(* CODESYS project Fiesto_workstation_Biraveen_Nedunchelian.export

Project tree, tasks and I/O mapping:
  Device : CODESYS Control Win V3 x64, 3S - Smart Software Solutions GmbH, version 3.5.16.30
    application Application
      libraries: Standard, * (System)
      task MainTask (cyclic, interval 50 ms, priority 1) calls PLC_PRG
      task VISU_TASK (cyclic, interval 100 ms, priority 31) calls VisuElems.Visu_Prg
      function block Festo_Workstation [ST]
      program PLC_PRG [CFC]
      visualisation Visualization
*)

// Device/Application/PLC_PRG
PROGRAM PLC_PRG
VAR
	Festo: Festo_Workstation;
	lav_indik10: BOOL;
	hoy_indik90: BOOL;
	tanknivaa_tank2: REAL;
	bryter: BOOL;
END_VAR

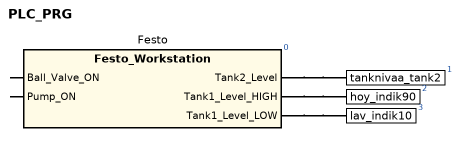
Festo(); // Festo_Workstation
tanknivaa_tank2 := Festo.Tank2_Level;
hoy_indik90 := Festo.Tank1_Level_HIGH;
lav_indik10 := Festo.Tank1_Level_LOW;

END_PROGRAM

// Device/Application/Festo_Workstation
FUNCTION_BLOCK Festo_Workstation
VAR_INPUT
	Ball_Valve_ON : BOOL := FALSE;
	Pump_ON : BOOL := FALSE;
END_VAR
VAR_OUTPUT
	Tank2_Level : REAL := 0;
	Tank1_Level_HIGH : BOOL := TRUE;
	Tank1_Level_LOW : BOOL := TRUE;
END_VAR
VAR
	Inflow : REAL := 0;
	Outflow : REAL := 0;
	Tank1_Level : REAL := 95;
	Inflow_Color : BOOL := FALSE;
	Outflow_Color : BOOL := FALSE;
	Reset : BOOL := FALSE;
	Av_var: REAL;
END_VAR

IF NOT Reset THEN //Reset er FALSE
	IF Pump_ON THEN //Er pumpen på?
		IF Tank1_Level > 0 THEN //Er det noe vann i tank 1? 
			Inflow := 0.2; //Fyll vann i tank 2
			Inflow_Color := TRUE; //Visuvar
		ELSE //Tank 1 er tom
			Inflow := 0; //Ikke fyll
			Inflow_Color := FALSE; //Visuvar
		END_IF
	ELSE //Pumpen er av
		Inflow := 0; //Ikke full
		Inflow_Color := FALSE; //Visuvar
	END_IF
	
	IF Ball_Valve_ON THEN //Er ventilen åpen
		IF Tank2_Level > 0 THEN //Er det vann i tank 2?
			Outflow := 0.1; //Det renner vann tilbake til tank 1
			Outflow_Color := TRUE; //Visuvar
		ELSE //Tank 2 er tom
			Outflow := 0; //Det renner ikke vann
			Outflow_Color := FALSE; //Visuvar
		END_IF
	ELSE //Ventilen er stengt
		Outflow := 0; //Det renner ikke vann
		Outflow_Color := FALSE; //Visuvar
	END_IF
	
	Tank1_Level := Tank1_Level + (Outflow - Inflow); //Level i tank 1
	Tank2_Level := Tank2_Level + (Inflow - Outflow); //Level i tank 2
	
	IF Tank1_Level >= 90 THEN //Er nivået i tank 1 større enn 90?
		Tank1_Level_HIGH := TRUE; //Variabelen er TRUE
	ELSE //Nivået er mindre enn 90
		Tank1_Level_HIGH := FALSE; //Variabel FALSE
	END_IF
	
	IF Tank1_Level <= 10 THEN //Er nivået i tank 1 mindre enn 10?
		Tank1_Level_LOW := FALSE; //Variabel FALSE
	ELSE //Nivået er større enn 10
		Tank1_Level_LOW := TRUE; //Variabel TRUE
	END_IF
ELSE //Reset er TRUE
	//Resetter variablene til initialverdier
	Inflow := 0;
	Outflow := 0;
	Tank1_Level := 95;
	Tank2_Level := 0;
	Tank1_Level_HIGH := FALSE;
	Tank1_Level_LOW := FALSE;
	Pump_ON := FALSE;
	Ball_Valve_ON := FALSE;
	Av_var := 0;
END_IF


IF Tank2_Level > 60 AND Av_var = 0 THEN
	Pump_ON := FALSE;
	Ball_Valve_ON := TRUE;
	Av_var := 1;
END_IF

IF Tank1_Level > 70 AND Av_var = 1 THEN
	Pump_ON := TRUE;
	Ball_Valve_ON := FALSE;
	Av_var := 2;
END_IF

IF Tank2_Level > 10 AND Av_var = 2 THEN
	Ball_Valve_ON := FALSE;
	Pump_ON := TRUE;
	Av_var := 0;
END_IF

END_FUNCTION_BLOCK

// Device/Application/Visualization
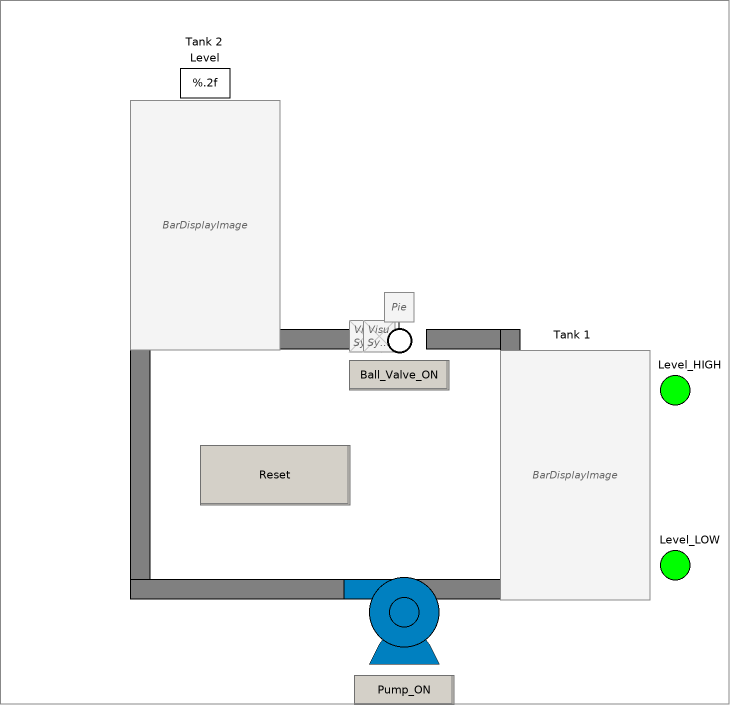
VISUALIZATION Visualization  // 730x705
    RoundedRectangle (426,329 86x20), colour toggle: PLC_PRG.Festo.Outflow_Color
    RoundedRectangle (500,329 20x30), colour toggle: PLC_PRG.Festo.Outflow_Color
    RoundedRectangle (275,329 96x20), colour toggle: PLC_PRG.Festo.Outflow_Color
    RoundedRectangle (130,338 20x260), colour toggle: PLC_PRG.Festo.Inflow_Color
    RoundedRectangle (355,579 150x20), colour toggle: PLC_PRG.Festo.Inflow_Color
    BarDisplayImage (130,100 150x250), value: PLC_PRG.Festo.Tank2_Level, style: BarDisplayImage-Gray, scale format: %.1f, scale 0..100
    BarDisplayImage (500,350 150x250), value: PLC_PRG.Festo.Tank1_Level, style: BarDisplayImage-Gray, scale format: %.1f, scale 0..100
    Group (335,577 104x87)
        Polygon (44,67) (69,34) (94,67) (104,87) (34,87)
        Rectangle (0,2 79x20)
        Ellipse (34,0 70x70)
        Ellipse (54,20 30x30)
    RoundedRectangle (130,579 214x20), colour toggle: PLC_PRG.Festo.Inflow_Color
    Group (349,292 100x68)
        Group (0,28 100x40)
            Image (0,0 32x32), image: VisuSymbols.Symbols.TriangleRight
            Image (14,0 32x32), image: VisuSymbols.Symbols.TriangleLeft
        Ellipse (38,36 25x25)
        Line (50,36) (50,16)
        Pie (35,0 30x30), angle 180
    Ellipse (660,550 30x30), colour toggle: PLC_PRG.Festo.Tank1_Level_LOW
        toggle PLC_PRG.lav_indik10
    Label (650,525 80x30), "Level_LOW"
    Ellipse (660,375 30x30), colour toggle: PLC_PRG.Festo.Tank1_Level_HIGH
        toggle PLC_PRG.hoy_indik90
    Label (650,350 80x30), "Level_HIGH"
    Rectangle (180,68 50x30), "%.2f", text variable: PLC_PRG.Festo.Tank2_Level
    Label (180,43 50x30), "Level"
    Button (349,360 100x30), "Ball_Valve_ON"
        toggle PLC_PRG.Festo.Ball_Valve_ON
    Button (354,675 100x30), "Pump_ON"
        toggle PLC_PRG.Festo.Pump_ON
    Button (200,445 150x60), "Reset"
        tap PLC_PRG.Festo.Reset
    Label (497,320 150x30), "Tank 1"
    Label (129,27 150x30), "Tank 2"
END_VISUALIZATION
